{attribute 'qualified_only'}
VAR_GLOBAL
    NC : AXIS_REF;
    MCS2 : AXIS_REF;
    E727 : AXIS_REF;
END_VAR

(* stored: Version 1.1.0.1
   GVL NcAxis_GVL: Id {20959dfc-4621-4990-a644-86123eb1a246} *)
